PROGRAM MAIN
VAR
END_VAR

END_PROGRAM

(* stored: Version 1.1.0.1
   POU MAIN: Id {921afc12-261a-4370-bb5b-70e9bb40d6bc} *)
